{attribute 'linkalways'} 
{attribute 'no_explicit_call' := 'This FB is a CLASS and must be accessed using methods or properties'}
{attribute 'enable_dynamic_creation'}
FUNCTION_BLOCK ABSTRACT MoveCommand EXTENDS AxisCommand IMPLEMENTS I_MoveCommand
VAR
	_velocity : LREAL;
	_acceleration: LREAL;
	_deceleration: LREAL;
	_jerk: LREAL;
	_bufferMode: AxisBufferMode;
END_VAR

END_FUNCTION_BLOCK

(* stored: Version 1.1.0.1, ProductVersion 3.1.4024.12
   POU MoveCommand: Id {965c49e3-202e-4ced-98b3-f8f941c0dc3b}, SpecialFunc None *)
